// TIA Portal project "创新任务+12452+12435" (V15.1)

(* hardware
DEVICE "S7-1200 station_1"  S7-1200 Station
   slot 0: "Rack_0"  S7-1200 Rack  Rack  V1.0
   slot 1: "PLC_1"  CPU 1212C DC/DC/DC  6ES7 212-1AE40-0XB0  V4.2
*)

// ===== PLC "PLC_1"  CPU 1212C DC/DC/DC =====

VAR_GLOBAL   // PLC tag table "默认变量表"
   "Tag_1" AT %I0.1 : Bool;
   "Tag_2" AT %M5.0 : Bool;
   "Tag_3" AT %M4.3 : Bool;
   "Tag_4" AT %M4.4 : Bool;
   "Tag_5" AT %M4.5 : Bool;
   "Tag_6" AT %M4.6 : Bool;
   "Tag_7" AT %M5.4 : Bool;
   "Tag_8" AT %Q0.0 : Bool;
   "Tag_9" AT %Q0.2 : Bool;
   "Tag_10" AT %Q0.1 : Bool;
END_VAR

// folder: System blocks/Program resources

DATA_BLOCK "c0"   // DB1
{ S7_Optimized_Access := 'TRUE' }
AUTHOR : Simatic
FAMILY : IEC
NAME : CNTR
VERSION : 1.0
// stored: InstanceOfName IEC_COUNTER
"IEC_COUNTER"
BEGIN
END_DATA_BLOCK

DATA_BLOCK "t3"   // DB3
{ S7_Optimized_Access := 'TRUE' }
AUTHOR : Simatic
FAMILY : IEC
NAME : IEC_TMR
VERSION : 1.0
// stored: InstanceOfName IEC_TIMER
"IEC_TIMER"
BEGIN
END_DATA_BLOCK

DATA_BLOCK "t4"   // DB4
{ S7_Optimized_Access := 'TRUE' }
AUTHOR : Simatic
FAMILY : IEC
NAME : IEC_TMR
VERSION : 1.0
// stored: InstanceOfName IEC_TIMER
"IEC_TIMER"
BEGIN
END_DATA_BLOCK

DATA_BLOCK "c3"   // DB5
{ S7_Optimized_Access := 'TRUE' }
AUTHOR : Simatic
FAMILY : IEC
NAME : CNTR
VERSION : 1.0
// stored: InstanceOfName IEC_COUNTER
"IEC_COUNTER"
BEGIN
END_DATA_BLOCK

// folder: (top level)

ORGANIZATION_BLOCK "Main"   // OB1, LAD, ProgramCycle
TITLE = "Main Program Sweep (Cycle)"
{ S7_Optimized_Access := 'TRUE' }
VERSION : 0.1
   VAR_INPUT
      Initial_Call : Bool;   // Initial call of this OB
      Remanence : Bool;   // =True, if remanent data are available
   END_VAR
BEGIN

REGION Network 1
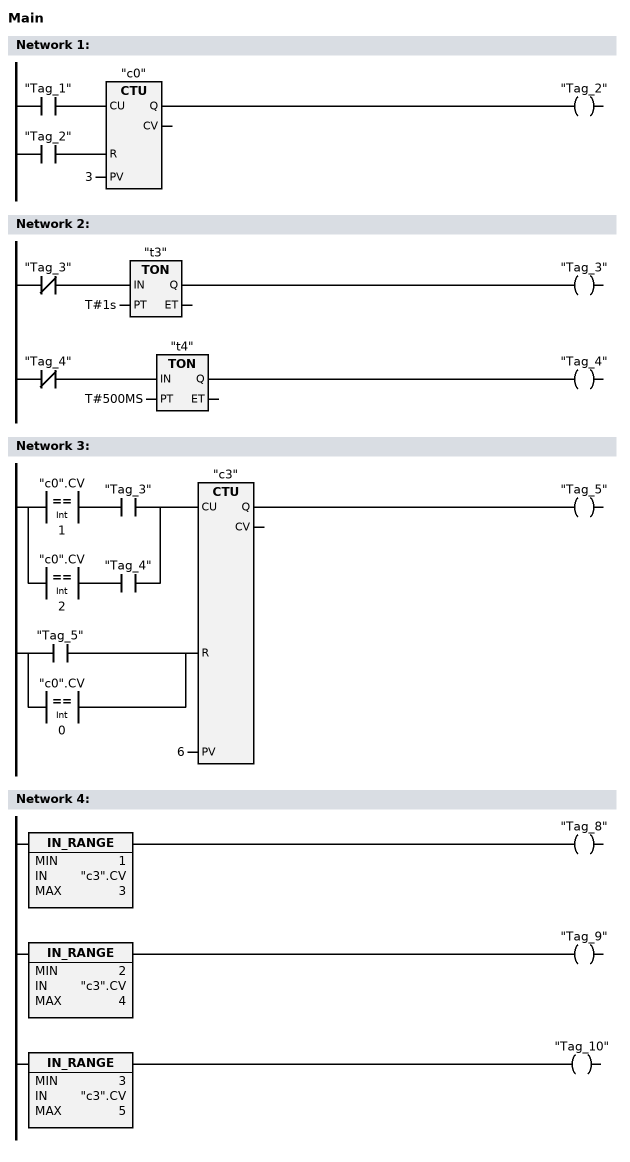
   "c0".CTU(CU := "Tag_1", R := "Tag_2", PV := 3);
   "Tag_2" := "c0".Q;
END_REGION

REGION Network 2
   "t3".TON(IN := NOT "Tag_3", PT := T#1s);
   "Tag_3" := "t3".Q;
   "t4".TON(IN := NOT "Tag_4", PT := T#500MS);
   "Tag_4" := "t4".Q;
END_REGION

REGION Network 3
   "c3".CTU(CU := (("c0".CV = 1) AND "Tag_3") OR (("c0".CV = 2) AND "Tag_4"),
            R := "Tag_5" OR ("c0".CV = 0),
            PV := 6);
   "Tag_5" := "c3".Q;
END_REGION

REGION Network 4
   RUNG wire#powerrail
      { S7_Templates := "SrcType := Int" } InRange(min := 1, in := "c3".CV, max := 3)
      Coil( "Tag_8" )
   END_RUNG
   RUNG wire#powerrail
      { S7_Templates := "SrcType := Int" } InRange(min := 2, in := "c3".CV, max := 4)
      Coil( "Tag_9" )
   END_RUNG
   RUNG wire#powerrail
      { S7_Templates := "SrcType := Int" } InRange(min := 3, in := "c3".CV, max := 5)
      Coil( "Tag_10" )
   END_RUNG
   // the same network as SCL:
   "Tag_8" := (1 <= "c3".CV) AND ("c3".CV <= 3);
   "Tag_9" := (2 <= "c3".CV) AND ("c3".CV <= 4);
   "Tag_10" := (3 <= "c3".CV) AND ("c3".CV <= 5);
END_REGION
END_ORGANIZATION_BLOCK